{attribute 'linkalways'} 
{attribute 'no_explicit_call' := 'This FB is a CLASS and must be accessed using methods or properties'}
{attribute 'enable_dynamic_creation'}
FUNCTION_BLOCK _ETcVnColorTrainingMethod EXTENDS EnumDatatypeBase
VAR
	localData : ETcVnColorTrainingMethod;
	activeData : REFERENCE TO ETcVnColorTrainingMethod;
	enumBaseDatatype : _DINT(localData);
END_VAR

METHOD PRIVATE AddLocalEnumeration
VAR_INPUT
	Enumeration : T_MAXSTRING;
	Value : ETcVnColorTrainingMethod;
END_VAR
AddEnumeration(Enumeration, Value);
END_METHOD

PROPERTY PUBLIC Address : PVOID
GET
Address := ADR(activeData);
END_GET
END_PROPERTY

METHOD PUBLIC ClearReference
VAR_INPUT
END_VAR
activeData REF= localData;
SetBaseDatatypeReference();
END_METHOD

METHOD PUBLIC Clone : I_Datatype
VAR
    pClone : POINTER TO _ETcVnColorTrainingMethod;
END_VAR
pClone := __NEW(_ETcVnColorTrainingMethod(InitialValue := Value));
Clone := pClone^;
END_METHOD

METHOD FB_init : BOOL
VAR_INPUT
	bInitRetains : BOOL; // if TRUE, the retain variables are initialized (warm start / cold start)
	bInCopyCode : BOOL;  // if TRUE, the instance afterwards gets moved into the copy code (online change)
	InitialValue : ETcVnColorTrainingMethod;
END_VAR
localData := InitialValue;
AddBaseDatatype(enumBaseDatatype);
ClearReference();

AddLocalEnumeration('TCVN_CTM_LAB', ETcVnColorTrainingMethod.TCVN_CTM_LAB);
AddLocalEnumeration('TCVN_CTM_RGB', ETcVnColorTrainingMethod.TCVN_CTM_RGB);
END_METHOD

PROPERTY PUBLIC Identifier : T_MAXSTRING
GET
Identifier := 'ETcVnColorTrainingMethod';
END_GET
END_PROPERTY

METHOD IsEnumeratorValueEqual : BOOL
VAR_INPUT
	Enumerator : I_KeyValueForwardEnumerator;
END_VAR
VAR
	storedValue : ETcVnColorTrainingMethod;
END_VAR
IF NOT Enumerator.TryGet(storedValue) THEN
	RETURN;
END_IF

IsEnumeratorValueEqual := storedValue = activeData;
END_METHOD

METHOD PUBLIC MakeReferenceTo
VAR_INPUT
	ReferenceTarget : REFERENCE TO ETcVnColorTrainingMethod;
END_VAR
activeData REF= ReferenceTarget;
SetBaseDatatypeReference();
END_METHOD

METHOD PROTECTED SetBaseDatatypeReference
VAR_INPUT
END_VAR
enumBaseDatatype.MakeReferenceTo(activeData);
END_METHOD

PROPERTY PUBLIC Size : UDINT
GET
Size := SIZEOF(activeData);
END_GET
END_PROPERTY

METHOD TryMakeReferenceTo : BOOL
VAR_INPUT
	Target : I_Datatype;
END_VAR
VAR
	targetAsEnum : I_EnumDatatype;
	pTargetData : POINTER TO ETcVnColorTrainingMethod;
END_VAR
IF NOT Target.TryResolveAsEnumDatatype(targetAsEnum) THEN
	RETURN;
END_IF

IF targetAsEnum.Identifier <> Identifier THEN
	RETURN;
END_IF

pTargetData := Target.Address;
activeData REF= pTargetData^;
SetBaseDatatypeReference();
TryMakeReferenceTo := TRUE;
END_METHOD

PROPERTY PUBLIC Value : ETcVnColorTrainingMethod
GET
Value := activeData;
END_GET
SET
activeData := Value;
END_SET
END_PROPERTY

END_FUNCTION_BLOCK

(* stored: Version 1.1.0.1
   POU _ETcVnColorTrainingMethod: Id {4120dfa5-bcd3-0c52-1c06-4232c1f35332}, SpecialFunc None
   Folder Constructor: Id {3abb8f7e-dc67-0e9e-0bb9-499de944dfce}
   Folder Private: Id {ee19857f-5805-0b8d-182c-62fd0bcc4a65}
   Folder Protected: Id {d01f5dc1-374d-0009-0ac0-d4dcbdee6115}
   Method AddLocalEnumeration: Id {96ebe17d-eedd-076d-0b96-e1e53da7ecc8}
   Property Address: Id {978a0e29-7b67-0543-1499-6811e955c738}
   Get Get: Id {bbdf0059-5d68-0206-3c90-b6b923804a95}
   Method ClearReference: Id {42878c02-396b-0428-3e8b-894ef798b261}
   Method Clone: Id {a3d36fc3-c196-027e-224b-06ab2aec6000}
   Method FB_init: Id {1488ff2d-9172-0925-2920-ae42a37506cd}
   Property Identifier: Id {2e1c9166-d7a2-0b19-2814-d29d75474ec6}
   Get Get: Id {5f32f7c8-604f-0572-08b2-d233263b4652}
   Method IsEnumeratorValueEqual: Id {7f15d113-7415-0c61-1939-05f3a40b721c}
   Method MakeReferenceTo: Id {cd679bbf-a9d8-0c50-0eb5-2a6554fdff89}
   Method SetBaseDatatypeReference: Id {57680102-40d7-0b2c-074c-a1e94e2dd655}
   Property Size: Id {b37cfa38-e3c2-07f1-2d07-fd7dd3570910}
   Get Get: Id {397fa90f-84d5-0d0c-16f9-a5971cd156f2}
   Method TryMakeReferenceTo: Id {dda1168e-4527-0950-3506-8650565e63bb}
   Property Value: Id {ae7d8133-eefe-0901-2623-922615c4ca55}
   Get Get: Id {76e99344-570a-0e1c-10ba-77958020e43d}
   Set Set: Id {bb600eeb-b7cf-034a-2d72-902f56f94481} *)
